TYPE E_ContactorControlMode :
(
    MANUAL := 0,        // Manuel kontrol - Lokal butonlar
    AUTO := 1,          // Otomatik kontrol - PLC lojiği
    REMOTE := 2         // Uzaktan kontrol - SCADA/HMI
);
END_TYPE

(* stored: Version 1.1.0.1, ProductVersion 3.1.4024.15
   EnumerationTextList E_ContactorControlMode: Id {87e58f04-4049-42ee-b036-b46d085a34a3} *)
